ABB RobotStudio station: Robot nailing.rsstn

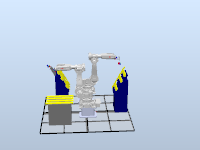
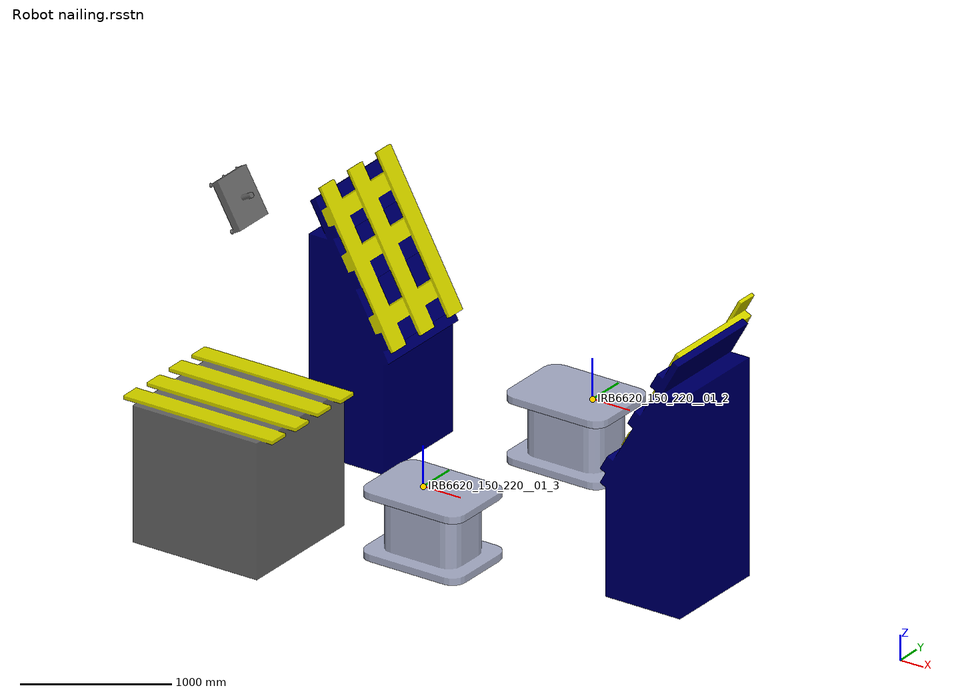
[picture v1: parts stored in the station drawn from their meshes, with robot base, taught points and paths (robot models come from the ABB library and are not in the file)]
Station Station (saved by RobotStudio 21.2.9526.0)
Controller Nailing, task T_ROB2: task frame (RAPID world) sits at (146.06, 1597.33, 476.12) mm in the station
Controller Nailing, task T_ROB1: task frame (RAPID world) sits at (146.06, 1597.33, 476.12) mm in the station
Controller Nailing
  mechanical unit ROB_1: IRB6620_150_220__01_2, 6 joints, base frame (0, -172.26, 0) mm
  mechanical unit ROB_2: IRB6620_150_220__01_3, 6 joints, base frame (-112.53, -1959.33, 41.86) mm, rotated rx 0 ry 0 rz 180 deg
Layout (positions relative to the parent item):
  - Palet_lucru [part] at (1605.21, 711.79, 1460.05) mm, rotated rx 61 ry 0 rz -90 deg, size 800 x 1200 x 80 mm
  - Palet_complet [part] at (-1039.1, 455.73, 1504.37) mm, rotated rx 61 ry 0 rz 90 deg, size 800 x 1200 x 80 mm
  - Tregaskiss22deg_rev0 [mechanism, from Tools\Tregaskiss_22deg.rslib] at (1526.26, 1425.08, 2231.12) mm, rotated rx 180 ry 60 rz 180 deg
  - piedestal_rs [part] at (28.69, 1403.02, 0) mm, size 800 x 600 x 500 mm
  - Suport_palet_5 [part] at (1952.51, -151.1, 798.88) mm, rotated rx 0 ry 0 rz 90 deg, size 801.1 x 643.6 x 1870.4 mm
  - Suport_palet_6 [part] at (-1417.49, 1195.73, 864.49) mm, rotated rx 0 ry 0 rz -90 deg, size 801.1 x 643.6 x 1870.4 mm
  - piedestal_rs_2 [part] at (79.78, -317.23, 0) mm, size 800 x 600 x 500 mm
  - IRB6620_150_220__01_2 [mechanism, from Robots\IRB6620_150_220_G_01.rslib] at (146.06, 1425.08, 476.12) mm; joint values [0, 0, 0, 0, 0.5236, 0] (rad or m)
  - IRB6620_150_220__01_3 [mechanism, from Robots\IRB6620_150_220_G_01.rslib] at (33.53, -361.99, 517.98) mm, rotated rx 0 ry 0 rz 180 deg; joint values [0, 0, 0, 0, 0.5236, 0] (rad or m)
  - Scandura [part] at (-1160.8, -904.27, 1001.19) mm, rotated rx 0 ry 0 rz 90 deg, size 150 x 1200 x 25 mm
  - Part_1 [part] at (-1668.92, -1270.41, 0) mm, size 1000 x 1000 x 1000 mm
  - Scandura_2 [part] at (-1178.12, -1147.63, 997.9) mm, rotated rx 0 ry 0 rz 90 deg, size 150 x 1200 x 25 mm
  - Scandura_3 [part] at (-1168.52, -374.66, 993.13) mm, rotated rx 0 ry 0 rz 90 deg, size 150 x 1200 x 25 mm
  - Scandura_3 [part] at (-1165.73, -642.32, 1002.28) mm, rotated rx 0 ry 0 rz 90 deg, size 150 x 1200 x 25 mm
  - Vacuum 2x3 [part] at (-1346.67, -361.99, 2272.98) mm, rotated rx 180 ry 60 rz 0 deg, size 372 x 332 x 160 mm
Attachment: Tregaskiss22deg_rev0 is attached to IRB6620_150_220__01_2 / Link6
Attachment: Vacuum 2x3 is attached to IRB6620_150_220__01_3 / Link6
EventTableEntry 1495: Group=, Trigger=vacuum 1496, Actions=[EventTableActionAttach 1497], Comment=, ActivationMode=2, Cyclic=false
EventTableTriggerIO 1496: IOValue=[1], IRC5Controller=? -1, Operator=0, SignalSource=Nailing 1503
EventTableActionAttach 1497: AttachmentParent=Vacuum 2x3 2518, AttachmentChild=? -1, MountObject=false, Offset=[X=1, Y=0, Z=0, W=0, X=0, Y=1, Z=0, W=0, X=0, Y=0, Z=1, W=0, X=0, Y=0, Z=0, W=1], FlangeIndext=0, FindNearest=true
EventTableEntry 1498: Group=, Trigger=vacuum 1499, Actions=[EventTableActionDetach 1500], Comment=, ActivationMode=2, Cyclic=false
EventTableTriggerIO 1499: IOValue=[0], IRC5Controller=? -1, Operator=0, SignalSource=Nailing 1503
EventTableActionDetach 1500: AttachmentParent=Vacuum 2x3 2518, AttachmentChild=? -1
Targets, tools, work objects and paths stored in the station, written as RAPID:
! task T_ROB1
MODULE CalibData
  PERS tooldata Tregaskiss22deg:=[TRUE,[[148.62,0.25,326.31],[0.833900724,0,0.551914471,0]],[1,[0,0,100],[1,0,0,0],0,0,0]];
ENDMODULE

! task T_ROB2
MODULE CalibData
  PERS tooldata Gripper_vacuum:=[TRUE,[[-248.167,-241.627,200.716],[1,0,0,0]],[10,[28.08,42.542,36.358],[1,0,0,0],0,0,0]];
ENDMODULE

